FUNCTION_BLOCK SampleComponentTests EXTENDS _internals_TcoContext
VAR
	_sut : TcoCognexVision.SampleComponent(THIS^);
END_VAR

{attribute 'TcRpcEnable'}
METHOD INTERNAL AddTwoNumbersTest : INT
VAR_INPUT
	NumberOne : INT;
	NumberTwo : INT;
END_VAR
AddTwoNumbersTest := _sut.AddTwoNumbers(NumberOne, NumberTwo);
END_METHOD

METHOD PROTECTED Main
END_METHOD

{attribute 'TcRpcEnable'}
METHOD INTERNAL WaitForModuloTest : BOOL
VAR_INPUT
	Modulo : INT;
END_VAR
WaitForModuloTest := _sut.WaitForModulo(Modulo);
END_METHOD

END_FUNCTION_BLOCK

(* stored: Version 1.1.0.1, ProductVersion 3.1.4024.9
   POU SampleComponentTests: Id {8976ba45-0863-0a6b-21c3-4f73a63db972}, SpecialFunc None
   Method AddTwoNumbersTest: Id {645d27ce-9e28-014e-310a-ae91dbed5602}
   Method Main: Id {72517ee4-edb7-004a-0cbc-276a16d1d561}
   Method WaitForModuloTest: Id {9c3fc460-8a59-0447-1fcb-e51f84ec6aef} *)
